{attribute 'qualified_only'}
VAR_GLOBAL
END_VAR

(* stored: Version 1.1.0.1, ProductVersion 3.1.4022.12
   GVL GVL_IO: Id {b8e7c4f4-3d10-4866-babb-7474574dffdf} *)
